PROGRAM POU
VAR
END_VAR

END_PROGRAM

(* stored: Version 1.1.0.1, ProductVersion 3.1.4024.9
   POU POU: Id {9538102e-97c9-49a7-877d-8f18a44c1d69}, SpecialFunc None *)
